FUNCTION_BLOCK SynchronizedAxisCommand EXTENDS AxisCommand IMPLEMENTS itfSynchronizedAxisCommand
VAR_INPUT
	_inSync	: REFERENCE TO BOOL;
END_VAR

PROPERTY InSync : BOOL
GET
InSync := _inSync;
END_GET
END_PROPERTY

END_FUNCTION_BLOCK

(* stored: Version 1.1.0.1, ProductVersion 3.1.4024.12
   POU SynchronizedAxisCommand: Id {fe2de06b-5354-4424-9064-414e3fd39de4}, SpecialFunc None
   Property InSync: Id {7688c86b-fa5d-4f2e-98b4-fa9c4c55dc1e}
   Get Get: Id {3f7abc23-1405-413c-9798-1e9c34d06acb} *)
